(* CODESYS project mobject-basic-nodepack.library
   Company: mobject
   DefaultNamespace: mobject-basic-nodepack
   Version: 0.4.0
   Placeholder: mobject-basic-nodepack
   Author: mobject dev team
   Title: mobject-basic-nodepack

Project tree, tasks and I/O mapping:
  libraries: mobject-basic-datatypes, 0.4.0 (mobject); mobject-datatypes, 0.7.0 (mobject); mobject-graph, 0.4.0 (mobject)
  Hardware/
    function block DigitalInputNode [ST]: FB_init, Clone, Dispose, OnExecute
    function block DigitalOutputNode [ST]: FB_init, Clone, Dispose, OnExecute
  function block BasicNodePack [ST]: RegisterWithNodeFactory
*)

// Hardware/DigitalInputNode
{attribute 'linkalways'} 
{attribute 'no_explicit_call' := 'This FB is a CLASS and must be accessed using methods or properties'}
{attribute 'enable_dynamic_creation'}
FUNCTION_BLOCK FINAL DigitalInputNode EXTENDS Node
VAR
	input AT %I* : BOOL;
	out : _BOOL(FALSE);
END_VAR

METHOD FB_init : BOOL
VAR_INPUT
	bInitRetains : BOOL; // if TRUE, the retain variables are initialized (warm start / cold start)
	bInCopyCode : BOOL;  // if TRUE, the instance afterwards gets moved into the copy code (online change)
END_VAR
AddOutput('out', out);
END_METHOD

METHOD PUBLIC Clone : I_Node
VAR
END_VAR
Clone := this^;
END_METHOD

METHOD Dispose
VAR_INPUT
END_VAR
END_METHOD

METHOD PROTECTED OnExecute : HRESULT
VAR
END_VAR
out.value := input;
END_METHOD

END_FUNCTION_BLOCK

// Hardware/DigitalOutputNode
{attribute 'linkalways'} 
{attribute 'no_explicit_call' := 'This FB is a CLASS and must be accessed using methods or properties'}
{attribute 'enable_dynamic_creation'}
FUNCTION_BLOCK FINAL DigitalOutputNode EXTENDS Node
VAR
	output AT %Q* : BOOL;
	in : _BOOL(FALSE);
END_VAR

METHOD FB_init : BOOL
VAR_INPUT
	bInitRetains : BOOL; // if TRUE, the retain variables are initialized (warm start / cold start)
	bInCopyCode : BOOL;  // if TRUE, the instance afterwards gets moved into the copy code (online change)
END_VAR
AddInput('in', in);
END_METHOD

METHOD PUBLIC Clone : I_Node
VAR
END_VAR
Clone := this^;
END_METHOD

METHOD Dispose
VAR_INPUT
END_VAR
END_METHOD

METHOD PROTECTED OnExecute : HRESULT
VAR
END_VAR
output := in.value;
END_METHOD

END_FUNCTION_BLOCK

// BasicNodePack
{attribute 'linkalways'} 
{attribute 'no_explicit_call' := 'This FB is a CLASS and must be accessed using methods or properties'}
{attribute 'enable_dynamic_creation'}
FUNCTION_BLOCK BasicNodePack IMPLEMENTS I_NodePack
VAR
END_VAR

METHOD PUBLIC RegisterWithNodeFactory
VAR_INPUT
	NodeFactory : I_NodeFactory;
END_VAR
END_METHOD

END_FUNCTION_BLOCK
